IF (count>=cTokenStringSetCount) THEN
	splitFQN := FALSE;
	RETURN;
END_IF
		
count := count + 1;
tokens[count] := MID(fqn,currentLength,position);

splitFQN := TRUE;

          
END_FUNCTION

FUNCTION_BLOCK TypeHandlerEnum EXTENDS TypeHandlerINT
  VAR CONSTANT
    cEnumOptionMax : USINT := 127;
  END_VAR
  VAR
    lDefinition : t_enum_option_definition;
    lFailed : BOOL := FALSE;
    lEnumOptionMax : USINT := 0;
    lEnumOptions : ARRAY[0..cEnumOptionMax] OF t_enum_option_definition;
  END_VAR

            
          

METHOD initialize
                  

                
END_METHOD

METHOD getValue : BOOL
  VAR_INPUT
    token : t_token_string;
    target : REFERENCE TO INT;
  END_VAR
  VAR
    i : USINT;
  END_VAR
                  FOR i:= 0 TO lEnumOptionMax DO
	IF (strcmp(token,lEnumOptions[i].token)) THEN
		getValue := TRUE;
		target := lEnumOptions[i].option;
		RETURN;
	END_IF
END_FOR

getValue := FALSE;

                
END_METHOD

METHOD getToken : t_token_string
  VAR_INPUT
    value : INT;
  END_VAR
  VAR
    index : USINT;
  END_VAR
                  index := mapping(value);

IF (index>lEnumOptionMax) THEN
	getToken := 'illegal';
	RETURN;
END_IF

getToken := lEnumOptions[index].token;

                
END_METHOD

METHOD defineOption
  VAR_INPUT
    option : INT;
    token : t_token_string;
    description : t_medium_string;
  END_VAR
  VAR
    ptr : POINTER TO t_enum_option_definition;
    index : USINT;
  END_VAR
                  index := mapping(option);

IF (index>cEnumOptionMax) THEN
	lFailed := TRUE;
	RETURN;
END_IF

lEnumOptionMax := MAX(lEnumOptionMax,index);

lEnumOptions[index].option := option;
lEnumOptions[index].token := token;
lEnumOptions[index].description := description;

                
END_METHOD

METHOD mapping : USINT
  VAR_INPUT
    option : INT;
  END_VAR
                  IF (lDefinition.option=cEnumTypeChannelMask) THEN
	mapping := 0;

	CASE option OF
	cChannelNone:
		mapping := 0;

	cChannelUIRadio:
		mapping := 1;

	cChannelUICabin:
		mapping := 2;

	cChannelLogTCP:
		mapping := 3;

	cChannelUIRCache:
		mapping := 4;

	cChannelMaster:
		mapping := 5;
		
	cChannelEdgeLog:
		mapping := 6;

	cChannelEdgeStateMetric:
		mapping := 7;

	cChannelEdgeValueMetric:
		mapping := 8;

	cChannelEdgeTrace:
		mapping := 9;
	END_CASE

	RETURN;
END_IF

IF (lDefinition.option=cEnumTypeDebugMask) THEN
	mapping := 0;

	CASE option OF
	cDebugNone:
		mapping := 0;

	cDebugWaitForLog:
		mapping := 1;

	cDebugEnableFailSafeOnCrash:
		mapping := 2;

	cDebugDisableWatchdog:
		mapping := 3;

	cDebugSimulateCrash:
		mapping := 4;

	cDebugSimulateA:
		mapping := 5;

	cDebugSimulateB:
		mapping := 6;

	cDebugSimulateC:
		mapping := 7;
	END_CASE

	RETURN;
END_IF

mapping :=INT_TO_USINT(option);
                
END_METHOD

METHOD getOptions : STRING
  VAR
    str : STRING;
    i : USINT;
    first : BOOL := TRUE;
  END_VAR
                  str := '[';

FOR i:=0 TO lEnumOptionMax DO
	IF (first) THEN
		str := CONCAT(str,'"');
		first := FALSE;
	ELSE
		str := CONCAT(str,', "');
	END_IF

	str := CONCAT(str,lEnumOptions[i].token);
	str := CONCAT(str,'"');
END_FOR

str := CONCAT(str,']');

getOptions := str;

                
END_METHOD

PROPERTY Definition : REFERENCE TO t_enum_option_definition
GET
                    Definition ref= lDefinition;
                  
END_GET
END_PROPERTY
END_FUNCTION_BLOCK
